{attribute 'GeneratedUsingTerminal: EL2911-0000-0016'}
{attribute addProperty BoxType "EL2911-0000-0016"}
{attribute addProperty Id "FSoE_CommandUSINT1FSOUT_Module_OutputBOOL1FSOUT_Module_ErrAckBOOL1FSIN_Module_ErrAckBOOL1FSoE_CRC_000UINT2FSoE_Connection_IDUINT2"}
{attribute addProperty CRC "3995974083"}
{attribute addProperty Size "8"}
TYPE FSOE_EE2DB9C3 :
STRUCT
	{attribute addProperty Name "FSoE_Command"}
	FSoE_Command : USINT;
	{attribute addProperty Name "FSOUT_Module_Output"}
	FSOUT_Module_Output : BOOL;
	{attribute addProperty Name "FSOUT_Module_ErrAck"}
	FSOUT_Module_ErrAck : BOOL;
	{attribute addProperty Name "FSIN_Module_ErrAck"}
	FSIN_Module_ErrAck : BOOL;
	{attribute addProperty Name "FSoE_CRC_000"}
	FSoE_CRC_000 : UINT;
	{attribute addProperty Name "FSoE_Connection_ID"}
	FSoE_Connection_ID : UINT;
END_STRUCT
END_TYPE

(* stored: Version 1.2.0.0, ProductVersion 3.1.4024.9
   DUT FSOE_EE2DB9C3: Id {faab8108-aa3c-4b46-8f5f-bcb57dec573d} *)
